TYPE Safety_Hmi :
STRUCT
	sStatusText			: Str;
	nStatusTextColor	: DWORD;
	
	bResetButton		: BOOL;
	bResetButtonVis		: BOOL;
END_STRUCT
END_TYPE

(* stored: Version 1.1.0.1
   DUT Safety_Hmi: Id {93f4fa20-c4bf-4746-b884-94b70b3e4255} *)
